// TIA Portal V15.1 export
// export: Created 2024-06-21T08:40:43.8494718Z, ExportSetting WithDefaults, DisplayName Totally Integrated Automation Portal, DisplayVersion V15.1 Update 5, DisplayName TIA Portal Openness, DisplayVersion V15.1 Update 5, DisplayName SINAMICS Startdrive Advanced, DisplayVersion V15.1, DisplayName G130, G150, S120, S150, SINAMICS MV, S210, DisplayVersion V15.1, DisplayName G110M, G120, G120C, G120D, G120P, DisplayVersion V15.1, DisplayName STEP 7 Professional, DisplayVersion V15.1 Update 5, DisplayName STEP 7 Safety, DisplayVersion V15.1, DisplayName WinCC Professional, DisplayVersion V15.1 Update 5, DisplayName SIMATIC Visualization Architect, DisplayVersion V15.1
DATA_BLOCK "_F209210ZS01Output"   // DB7012, F_DB
{ S7_Optimized_Access := 'TRUE' }
VERSION : 0.1
// stored: AutoNumber false, DBAccessibleFromOPCUA true
   VAR
      "209000AK03F9QC1FbkError" { ExternalAccessible := 'False'; ExternalVisible := 'False'; ExternalWritable := 'False'} : Bool;   // 210CR21 Feedback Error Brake 400VAC OFF -> contactor QC1
      "209000AK03F9QC2FbkError" { ExternalAccessible := 'False'; ExternalVisible := 'False'; ExternalWritable := 'False'} : Bool;   // 210CR21 Feedback Error Brake 400VAC OFF -> contactor QC2
      "209000AK03F9QC3FbkError" { ExternalAccessible := 'False'; ExternalVisible := 'False'; ExternalWritable := 'False'} : Bool;   // 210CS22 Feedback Error Brake 400VAC OFF -> contactor QC3
      "209000AK03F9QC4FbkError" { ExternalAccessible := 'False'; ExternalVisible := 'False'; ExternalWritable := 'False'} : Bool;   // 210CS22 Feedback Error Brake 400VAC OFF -> contactor QC4
      "209000AK03F9QC5FbkError" { ExternalAccessible := 'False'; ExternalVisible := 'False'; ExternalWritable := 'False'} : Bool;   // 210CR23 Feedback Error Brake 400VAC OFF -> contactor QC5
      "209000AK03F9QC6FbkError" { ExternalAccessible := 'False'; ExternalVisible := 'False'; ExternalWritable := 'False'} : Bool;   // 210CR23 Feedback Error Brake 400VAC OFF -> contactor QC6
   END_VAR
BEGIN
END_DATA_BLOCK
